// TIA Portal V20 export
// export: Created 2025-12-01T14:57:28.2232406Z, ExportSetting None, DisplayName Totally Integrated Automation Portal, DisplayVersion V20 Update 3, DisplayName TIA Portal Openness, DisplayVersion V20 Update 3, DisplayName TIA Portal Version Control Interface, DisplayVersion V20 Update 3, DisplayName STEP 7 Professional, DisplayVersion V20 Update 3, DisplayName STEP 7 Safety, DisplayVersion V20 Update 2, DisplayName WinCC Basic/Comfort/Advanced, DisplayVersion V20 Update 3, DisplayName WinCC Professional, DisplayVersion V20 Update 3, DisplayName WinCC Unified, DisplayVersion V20 Update 3
FUNCTION_BLOCK "FB605_SalidaFija_Quimarox"   // FB605, LAD
{ S7_Optimized_Access := 'FALSE' }
// stored: AutoNumber false, SetENOAutomatically false
   VAR_INPUT
      MesaSiguiente : UInt;
      MesaDeDescarga : UInt;
      ID_Quimarox : UInt;
      ID_Elemento : UInt;
      EnTension : Bool;
      Termico : Bool;
      pHs_PosicionDescarga : Bool;
      pHs_Protrusion : Bool;
      NXT_PTF : Bool;
      NXT_FTF : Bool;
      V_FILTRO_pHsPresencia : Int;
      Pto_Ajuste_1 : Int;   // Error_protusion
      Pto_Ajuste_2 : Int;   // Paso_A_Lenta
      Pto_Ajuste_3 : Int;   // Error_protusion
   END_VAR
   VAR_OUTPUT
      NXT_DescargaActiva : Bool;   // permiso mesa anterior y avance de la siguiente
      NXT_AVTF : Bool;
      PararElevador : Bool;
      ElevadorEnLenta : Bool;
      Avance_SalidaFija : Bool;
   END_VAR
   VAR
      TMP_EnTension { S7_SetPoint := 'True'} : "FB910_CNT_UHS";
      FILTRO_pHsPresencia { S7_SetPoint := 'True'} : "FB910_CNT_UHS";
      EstadoAsociadoEnMesa { S7_SetPoint := 'True'} : UInt;
      Aux_PeineEnDesCarga : UInt;
      PresenciaEnReset : Bool;
   END_VAR
   VAR_TEMP
      TMP_PeineDeCarga : UInt;
      MesaQuimarox : UInt;
      NumeroUT : UInt;
      EsMesaTL : Bool;
      FILTRO_PosicionDesCarga : Bool;
   END_VAR
BEGIN

NETWORK
TITLE = ERROR - Rearme
/////////////////////////////////////////////////////////////
/////////////////////////////////////////////////////////////
/////////////////////////////////////////////////////////////
// Rearne de Errores
      SET;
      A     "DB902_Estado_ZonaMesa".EstadoMesas[#MesaDeDescarga].Rearme_CBx;
      O     "DB902_Estado_ZonaMesa".EstadoMesas[#MesaDeDescarga].PerReset_CBx;
      R     "DB900_Estado_Mesas".EstadoVI[#MesaDeDescarga].Error_Mx;
      R     "DB900_Estado_Mesas".EstadoVI[#MesaDeDescarga].Err_Protusion;
      R     "DB900_Estado_Mesas".EstadoVI[#MesaDeDescarga].Err_DatosPLC;
      R     "DB900_Estado_Mesas".EstadoVI[#MesaDeDescarga].Err_Termico_E1_E3;
      R     "DB900_Estado_Mesas".EstadoVI[#MesaDeDescarga].Err_Perdida_PHs;


NETWORK
TITLE = RECEP OK DE LA ORDEN -- NO SE UTILIZA
/////////////////////////////////////////////////////////////
/////////////////////////////////////////////////////////////
/////////////////////////////////////////////////////////////
// RECEP OK DE LA ORDEN
      SET;
      AN    "DB841_Recepcion".Mesa[#MesaDeDescarga].Protocolo.Ord_S00;
      AN    "DB841_Recepcion".Mesa[#MesaDeDescarga].Protocolo.Ord_S01;
      AN    "DB841_Recepcion".Mesa[#MesaDeDescarga].Protocolo.Ord_S02;
      AN    "DB841_Recepcion".Mesa[#MesaDeDescarga].Protocolo.Ord_S03;
      NOT;
      =     "DB840_Emision".Mesa[#MesaDeDescarga].Protocolo.RecepOK;



NETWORK
TITLE = HMI - Manual
/////////////////////////////////////////////////////////////
/////////////////////////////////////////////////////////////
/////////////////////////////////////////////////////////////
// Para HMI >>> Manual
      SET;
      O     "DB902_Estado_ZonaMesa".EstadoMesas[#MesaDeDescarga].Manual_CBx;
      =     "DB900_Estado_Mesas".EstadoVI[#MesaDeDescarga].Manual;



NETWORK
TITLE = HMI - Entradas y Salidas de la Mesa
/////////////////////////////////////////////////////////////
/////////////////////////////////////////////////////////////
/////////////////////////////////////////////////////////////
// Entradas
      SET;
      A     #pHs_PosicionDescarga;
      =     "DB900_Estado_Mesas".EstadoVI[#MesaDeDescarga].En_PHS_1;
      SET;
      A     #pHs_Protrusion;
      =     "DB900_Estado_Mesas".EstadoVI[#MesaDeDescarga].En_pHs_Prot1;

      SET;
      A     #Termico;
      =     "DB900_Estado_Mesas".EstadoVI[#MesaDeDescarga].En_Termico1;


// Salidas
      SET;
      A     #Avance_SalidaFija;
      =     "DB900_Estado_Mesas".EstadoVI[#MesaDeDescarga].Sa_Rod_Avance;



NETWORK
TITLE = Comprobacion de que la MESA es de TRACKING
/////////////////////////////////////////////////////////////
/////////////////////////////////////////////////////////////
/////////////////////////////////////////////////////////////
// Comprobar si es una Mesa de Tracking o Routing
      SET;
      A     "DB850_DefinicionMesas".Mesa[#MesaDeDescarga].ConfigMesa.MesaTL;
      =     #EsMesaTL;



REGION Network 6: TMP - Espera En Tension
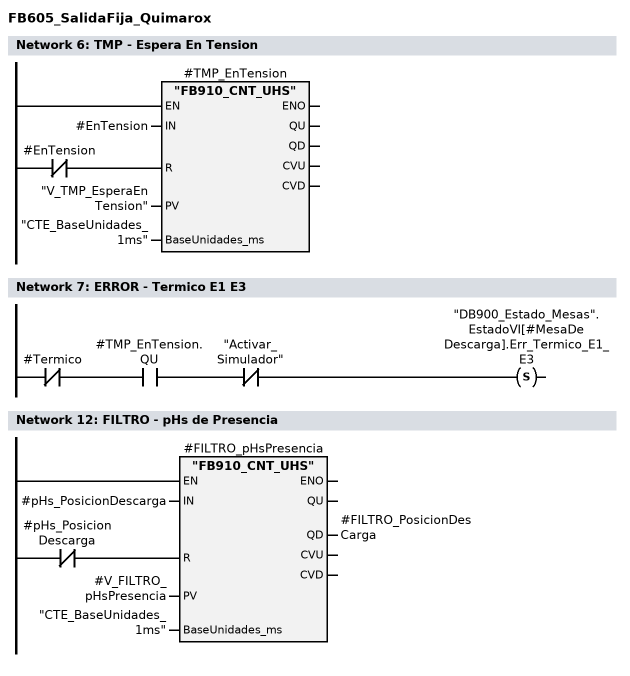
   RUNG wire#powerrail
      #TMP_EnTension(R := wire#w1, IN := #EnTension, PV := "V_TMP_EsperaEnTension", BaseUnidades_ms := "CTE_BaseUnidades_1ms", QU =>, QD =>, CVU =>, CVD =>)
   END_RUNG
   RUNG wire#powerrail
      I_Contact( #EnTension )
   END_RUNG wire#w1
   // the same network as SCL:
   #TMP_EnTension(IN := #EnTension,   // "FB910_CNT_UHS"
                  R := NOT #EnTension,
                  PV := "V_TMP_EsperaEnTension",
                  BaseUnidades_ms := "CTE_BaseUnidades_1ms");
END_REGION

REGION Network 7: ERROR - Termico E1 E3
   RUNG wire#powerrail
      I_Contact( #Termico )
      Contact( #TMP_EnTension.QU )
      I_Contact( "Activar_Simulador" )
      S_Coil( "DB900_Estado_Mesas".EstadoVI[#MesaDeDescarga].Err_Termico_E1_E3 )
   END_RUNG
   // the same network as SCL:
   IF NOT #Termico AND #TMP_EnTension.QU AND NOT "Activar_Simulador" THEN
       "DB900_Estado_Mesas".EstadoVI[#MesaDeDescarga].Err_Termico_E1_E3 := TRUE;
   END_IF;
END_REGION

NETWORK
TITLE = INICIALIZACION Previa
/////////////////////////////////////////////////////////////
/////////////////////////////////////////////////////////////
/////////////////////////////////////////////////////////////
      CLR;
      =     #NXT_DescargaActiva;
      =     #NXT_AVTF;

      CLR;
      =     #ElevadorEnLenta;
      =     #PararElevador;
      =     #Avance_SalidaFija;

      CLR;
      =     "DB900_Estado_Mesas".EstadoVI[#MesaDeDescarga].Etapas_Reset;
      =     "DB900_Estado_Mesas".EstadoVI[#MesaDeDescarga].Etapa_Vacia;
      =     "DB900_Estado_Mesas".EstadoVI[#MesaDeDescarga].Etapa_Cargada;
      =     "DB900_Estado_Mesas".EstadoVI[#MesaDeDescarga].Etapas_Carga_E0;
      =     "DB900_Estado_Mesas".EstadoVI[#MesaDeDescarga].Etapas_Descarga_S3;



NETWORK
TITLE = SISTEMA - Paro Blando
/////////////////////////////////////////////////////////////
/////////////////////////////////////////////////////////////
/////////////////////////////////////////////////////////////
// - Inicializar Variables de PARO BLANDO
      CLR;
      =     "DB900_Estado_Mesas".EstadoVI[#MesaDeDescarga].Paro_Blando;

/////////////////////////////////////////////////////////////
// - Existe PARO BLANDO ???
      SET;
      AN    "DB902_Estado_ZonaMesa".EstadoMesas[#MesaDeDescarga].ParoBlando_CBx;
      JC    NoRealizandose_ParoBlando;

/////////////////////////////////////////////////////////////
// - Fin de PARO BLANDO
      SET;
      =     "DB900_Estado_Mesas".EstadoVI[#MesaDeDescarga].Paro_Blando;


/////////////////////////////////////////////////////////////
/////////////////////////////////////////////////////////////
/////////////////////////////////////////////////////////////
// - Final Tratamiento del PARO BLANDO
NoRealizandose_ParoBlando:NOP   0;



NETWORK
TITLE = SISTEMA - Reset
/////////////////////////////////////////////////////////////
/////////////////////////////////////////////////////////////
/////////////////////////////////////////////////////////////
// -- Inicializar Variables de RESET
      SET;
      AN    "DB902_Estado_ZonaMesa".EstadoMesas[#MesaDeDescarga].PerReset_CBx;
      R     "DB900_Estado_Mesas".EstadoVI[#MesaDeDescarga].Fin_VI;
      R     #PresenciaEnReset;

/////////////////////////////////////////////////////////////
/////////////////////////////////////////////////////////////
/////////////////////////////////////////////////////////////
// - Existe RESET ??
      SET;
      AN    "DB902_Estado_ZonaMesa".EstadoMesas[#MesaDeDescarga].PerReset_CBx;
      JC    NoRealizandose_Reset;

      L     0;  // Estado de La Mesa = 0
      T     #EstadoAsociadoEnMesa;
      SET;
      =     "DB900_Estado_Mesas".EstadoVI[#MesaDeDescarga].Etapas_Reset;

/////////////////////////////////////////////////////////////
/////////////////////////////////////////////////////////////
/////////////////////////////////////////////////////////////
// - Emision de Presencia en caso de Reset
      SET;  // Presencia >>> Reset Total
      A     #pHs_PosicionDescarga;
      A     "DB831_Mesas".Mesas[#MesaDeDescarga].Memorias.M_ResetTotal;
      AN    #PresenciaEnReset;
      JC    Enviar_PresenciaEnResetTotal;

      SET;  // Presencia >>> Reset Parcial
      A     #pHs_PosicionDescarga;
      A     "DB831_Mesas".Mesas[#MesaDeDescarga].Memorias.M_ResetParcial;
      AN    #PresenciaEnReset;
      JC    Enviar_PresenciaEnResetParcial;

      JU    Final_PresenciaEnReset;

// - Presencia en Reset TOTAL >>> Enviar NUUT
Enviar_PresenciaEnResetTotal:NOP   0;
      CALL  "FC723_InsertarUT_EnMesa"
      ( MesaActual := #MesaDeDescarga,
        NumeroUT   := #NumeroUT
      );
      L     132;  // Envio de Nueva UT en RESET
      T     "DB812_UTs_Control".UT[#NumeroUT].EstadoEventoAGenerar;

      SET;  // Ya esta Avisado el JdT
      S     #PresenciaEnReset;

      JU    Final_PresenciaEnReset;

// - Presencia en Reset Parcial >>> Enviar LOCA en Reset Pantalla
Enviar_PresenciaEnResetParcial:NOP   0;
      L     "DB810_ColasMesas".Colas[#MesaDeDescarga].UT_PrimeraMesa;
      T     #NumeroUT;

      L     #NumeroUT;  // Comprobar que Existe UT
      L     0;
      ==I;
      JC    ErrorDatosCargada;

      L     101;  // Envio de LOCA en RESET
      T     "DB812_UTs_Control".UT[#NumeroUT].EstadoEventoAGenerar;

      SET;  // Ya esta Avisado el JdT
      S     #PresenciaEnReset;

      JU    Final_PresenciaEnReset;

// - Final de la Presencia En Reset
Final_PresenciaEnReset:NOP   0;


/////////////////////////////////////////////////////////////
/////////////////////////////////////////////////////////////
/////////////////////////////////////////////////////////////
// - Fin de RESET
      SET;  // Con Presencia de Carga >>> TOTAL
      A(;
      L     "DB810_ColasMesas".Colas[#MesaDeDescarga].UT_PrimeraMesa;
      L     0;
      ==I;
      );
      A     #pHs_PosicionDescarga;
      A     #PresenciaEnReset;
      A     "DB831_Mesas".Mesas[#MesaDeDescarga].Memorias.M_ResetTotal;
      S     "DB900_Estado_Mesas".EstadoVI[#MesaDeDescarga].Fin_VI;

      SET;  // Con Presencia de Carga >>> PARCIAL
      A     #pHs_PosicionDescarga;
      A     #PresenciaEnReset;
      A     "DB831_Mesas".Mesas[#MesaDeDescarga].Memorias.M_ResetParcial;
      S     "DB900_Estado_Mesas".EstadoVI[#MesaDeDescarga].Fin_VI;


      SET;  // Sin Presencia de Carga
      AN    #pHs_PosicionDescarga;
      S     "DB900_Estado_Mesas".EstadoVI[#MesaDeDescarga].Fin_VI;

      BE;

/////////////////////////////////////////////////////////////
/////////////////////////////////////////////////////////////
/////////////////////////////////////////////////////////////
// - Final Tratamiento del RESET
NoRealizandose_Reset:NOP   0;



NETWORK
TITLE = >>>>>>>>>>>>>>>>>>>>>>>>>>>>>>>>>>>>>>>>>>>>>>>>>>>>>>>>>>>>>>>>>>>

REGION Network 12: FILTRO - pHs de Presencia
   RUNG wire#powerrail
      #FILTRO_pHsPresencia(R := wire#w1, IN := #pHs_PosicionDescarga, PV := #V_FILTRO_pHsPresencia, BaseUnidades_ms := "CTE_BaseUnidades_1ms", QU =>, QD => #FILTRO_PosicionDesCarga, CVU =>, CVD =>)
   END_RUNG
   RUNG wire#powerrail
      I_Contact( #pHs_PosicionDescarga )
   END_RUNG wire#w1
   // the same network as SCL:
   #FILTRO_pHsPresencia(IN := #pHs_PosicionDescarga,   // "FB910_CNT_UHS"
                        R := NOT #pHs_PosicionDescarga,
                        PV := #V_FILTRO_pHsPresencia,
                        BaseUnidades_ms := "CTE_BaseUnidades_1ms",
                        QD => #FILTRO_PosicionDesCarga);
END_REGION

NETWORK
TITLE = >>>>>>>>>>>>>>>>>>>>>>>>>>>>>>>>>>>>>>>>>>>>>>>>>>>>>>>>>>>>>>>>>>>

NETWORK
TITLE = DISTRIBUCION >>> Control Etapa Activa
/////////////////////////////////////////////////////////////////////////////////////
/////////////////////////////////////////////////////////////////////////////////////
/////////////////////////////////////////////////////////////////////////////////////
// -- Listado de saltos de programa  >>> Estado
      L     #EstadoAsociadoEnMesa;
      JL    ESTADO_PorDefecto;

      JU    ETAPA_00_EnReset;
      JU    ETAPA_01_EnReposo;
      JU    ETAPA_02_EsperaDesCarga;
      JU    ETAPA_03_DesCargando;
      JU    ETAPA_04_FinalDeDescarga;

      JU    ESTADO_PorDefecto;
      JU    ESTADO_PorDefecto;
      JU    ESTADO_PorDefecto;
      JU    ESTADO_PorDefecto;
      JU    ESTADO_PorDefecto;

      JU    ETAPA_10_ResetCargado_EsperaDesCarga;
      JU    ETAPA_11_ResetCargado_DesCargando;
      JU    ETAPA_12_ResetCargado_FinalDeDescarga;

ESTADO_PorDefecto:JU    FinalFuncion;



NETWORK
TITLE = ETAPA 00 >>> En Reset
/////////////////////////////////////////////////////////////////////////////////////
/////////////////////////////////////////////////////////////////////////////////////
/////////////////////////////////////////////////////////////////////////////////////
ETAPA_00_EnReset:NOP   0;
      SET;
      =     "DB900_Estado_Mesas".EstadoVI[#MesaDeDescarga].Etapas_Reset;

/////////////////////////////////////////////////////////////////////////////////////
// generación de error de protusion
      SET;
      AN    #pHs_Protrusion;
      JC    ErrorProtrusion;


/////////////////////////////////////////////////////////////////////////////////////
// Tiene que estar en Marcha y Sin Error para continuar
      SET;
      AN    "DB902_Estado_ZonaMesa".EstadoMesas[#MesaDeDescarga].Marcha_CBx;
      O     "DB902_Estado_ZonaMesa".EstadoMesas[#MesaDeDescarga].Error_CBx;
      JC    ET00_PararElevador;


/////////////////////////////////////////////////////////////////////////////////////
// Sin Carga
      SET;
      AN    #FILTRO_PosicionDesCarga;
      JC    ET00_IrEtapa_01_EnReposo;

// Con Carga
      SET;
      A     #FILTRO_PosicionDesCarga;
      JC    ET00_IrEtapa_10_ResetCargado_EsperaDesCarga;
      BE;


/////////////////////////////////////////////////////////////////////////////////////
/////////////////////////////////////////////////////////////////////////////////////
/////////////////////////////////////////////////////////////////////////////////////
ET00_PararElevador:NOP   0;
      SET;
      =     #PararElevador;
      BE;


/////////////////////////////////////////////////////////////////////////////////////
/////////////////////////////////////////////////////////////////////////////////////
/////////////////////////////////////////////////////////////////////////////////////
ET00_IrEtapa_01_EnReposo:NOP   0;
      L     1;
      T     #EstadoAsociadoEnMesa;
      JU    ETAPA_01_EnReposo;


/////////////////////////////////////////////////////////////////////////////////////
/////////////////////////////////////////////////////////////////////////////////////
/////////////////////////////////////////////////////////////////////////////////////
ET00_IrEtapa_10_ResetCargado_EsperaDesCarga:NOP   0;
      SET;  // No existe UT >>> Error de Datos
      A(;
      L     "DB810_ColasMesas".Colas[#MesaDeDescarga].UT_PrimeraMesa;
      L     0;
      ==I;
      );
      AN    #EsMesaTL;
      JC    ErrorDatosCargada;

      L     10;
      T     #EstadoAsociadoEnMesa;
      JU    ETAPA_10_ResetCargado_EsperaDesCarga;



NETWORK
TITLE = ETAPA 01 >>> En Reposo
/////////////////////////////////////////////////////////////////////////////////////
/////////////////////////////////////////////////////////////////////////////////////
/////////////////////////////////////////////////////////////////////////////////////
// comprobamos si tenemos que parar el elevador por seguridad
ETAPA_01_EnReposo:NOP   0;
      SET;
      =     "DB900_Estado_Mesas".EstadoVI[#MesaDeDescarga].Etapa_Vacia;


/////////////////////////////////////////////////////////////////////////////////////
// Comprobar si hay algo en la Mesa
      SET;
      A     #FILTRO_PosicionDesCarga;
      JC    ET01_IrEtapa_02_SalidaDePeine;

/////////////////////////////////////////////////////////////////////////////////////
/////////////////////////////////////////////////////////////////////////////////////
/////////////////////////////////////////////////////////////////////////////////////
// error protusion, hay algo y en ese momento no debería haber nada
      SET;
      AN    "DB602_ElementosQuimarox".Quimarox[#ID_Quimarox].Elementos[#ID_Elemento].Hay_Carrier_en_ventana;
      A(;
      ON    #pHs_Protrusion;
      O     #FILTRO_PosicionDesCarga;
      );
      JC    ErrorProtrusion;

/////////////////////////////////////////////////////////////////////////////////////
// error protusion, hay algo y en ese momento no debería haber nada
      SET;
      A     "DB602_ElementosQuimarox".Quimarox[#ID_Quimarox].Elementos[#ID_Elemento].Hay_Carrier_en_ventana;
      A(;
      L     "DB602_ElementosQuimarox".Quimarox[#ID_Quimarox].Elementos[#ID_Elemento].Avance_carrier;
      L     #Pto_Ajuste_1;
      <=I;
      );
      A(;
      ON    #pHs_Protrusion;
      O     #FILTRO_PosicionDesCarga;
      );
      JC    ErrorProtrusion;


/////////////////////////////////////////////////////////////////////////////////////
/////////////////////////////////////////////////////////////////////////////////////
/////////////////////////////////////////////////////////////////////////////////////
// No deberia estar en este Estado, ha pasado sin carga


/////////////////////////////////////////////////////////////////////////////////////
// Parar por seguridad
      SET;
      A     "DB602_ElementosQuimarox".Quimarox[#ID_Quimarox].Elementos[#ID_Elemento].Hay_Carrier_en_ventana;
      A(;
      L     "DB602_ElementosQuimarox".Quimarox[#ID_Quimarox].Elementos[#ID_Elemento].Avance_carrier;  // #datos_elemento_Tmp.Avance_carrier
      L     #Pto_Ajuste_3;
      >=I;
      );
      A(;
      ON    #pHs_Protrusion;
      O     #FILTRO_PosicionDesCarga;
      );
      JC    ET01_PararElevador;


/////////////////////////////////////////////////////////////////////////////////////
// Lenta por seguridad
      SET;
      A     "DB602_ElementosQuimarox".Quimarox[#ID_Quimarox].Elementos[#ID_Elemento].Hay_Carrier_en_ventana;
      A(;
      L     "DB602_ElementosQuimarox".Quimarox[#ID_Quimarox].Elementos[#ID_Elemento].Avance_carrier;  // #datos_elemento_Tmp.Avance_carrier
      L     #Pto_Ajuste_2;
      >=I;
      );
      A(;
      ON    #pHs_Protrusion;
      O     #FILTRO_PosicionDesCarga;
      );
      JC    ET01_VelocidadLenta;

/////////////////////////////////////////////////////////////////////////////////////
// Final de Estado
      BE;


/////////////////////////////////////////////////////////////////////////////////////
/////////////////////////////////////////////////////////////////////////////////////
/////////////////////////////////////////////////////////////////////////////////////
ET01_PararElevador:NOP   0;
      SET;
      =     #PararElevador;

      BE;

/////////////////////////////////////////////////////////////////////////////////////
/////////////////////////////////////////////////////////////////////////////////////
/////////////////////////////////////////////////////////////////////////////////////
ET01_VelocidadLenta:NOP   0;
      SET;
      =     #ElevadorEnLenta;
      BE;


/////////////////////////////////////////////////////////////////////////////////////
/////////////////////////////////////////////////////////////////////////////////////
/////////////////////////////////////////////////////////////////////////////////////
ET01_IrEtapa_02_SalidaDePeine:NOP   0;
      L     "DB602_ElementosQuimarox".Quimarox[#ID_Quimarox].Elementos[#ID_Elemento].Numero_carrier;
      T     #Aux_PeineEnDesCarga;

// Emision del Evento del Quimarox
      L     "CTE_Evento_QDES";
      T     "DB601_PeinesQuimarox".Quimarox[#ID_Quimarox].vagon[#Aux_PeineEnDesCarga].EventoAGenerar;
      L     #MesaDeDescarga;
      L     "CTE_OffsetMesa";
      +I;
      T     "DB601_PeinesQuimarox".Quimarox[#ID_Quimarox].vagon[#Aux_PeineEnDesCarga].Mesa_descarga;

/////////////////////////////////////////////////////////////////////////////////////
/////////////////////////////////////////////////////////////////////////////////////
/////////////////////////////////////////////////////////////////////////////////////
// Comprobar Tipo de Mesa
      SET;
      A     #EsMesaTL;
      JC    ET01_Final_RecogerDatosDelPeine;

/////////////////////////////////////////////////////////////////////////////////////
// TRACKING - INICIO - Recoger Datos del Peine
      SET;
      L     "DB601_PeinesQuimarox".Quimarox[#ID_Quimarox].vagon[#Aux_PeineEnDesCarga].DatosCarga.Mckey;
      L     0;
      ==D;
      JC    ET01_TRACKING_CrearNueva_UT;
      JU    ET01_TRACKING_Crear_UT;


/////////////////////////////////////////////////////////////////////////////////////
// TRAKING - NuevaUT en la Mesa
ET01_TRACKING_Crear_UT:NOP   0;
      CALL  "FC721_CrearUT_EnMesa"
      ( McKey      := "DB601_PeinesQuimarox".Quimarox[#ID_Quimarox].vagon[#Aux_PeineEnDesCarga].DatosCarga.Mckey,
        MesaActual := #MesaDeDescarga,
        NumeroUT   := #NumeroUT
      );

      L     100;  // Emitir evento LOCA
      T     "DB812_UTs_Control".UT[#NumeroUT].EstadoEventoAGenerar;

      L     "DB601_PeinesQuimarox".Quimarox[#ID_Quimarox].vagon[#Aux_PeineEnDesCarga].DatosCarga.MesaDestino;
      T     "DB812_UTs_Control".UT[#NumeroUT].MesaDestino;
      T     "DB812_UTs_Control".UT[#NumeroUT].MesaIntermedia;
      T     "DB813_UTs_Ruta".UT[#NumeroUT].Ruta[0];

      JU    ET01_Final_RecogerDatosDelPeine;


/////////////////////////////////////////////////////////////////////////////////////
// TRAKING - NuevaUT en la Mesa
ET01_TRACKING_CrearNueva_UT:NOP   0;
      JU    ET01_Final_RecogerDatosDelPeine;


/////////////////////////////////////////////////////////////////////////////////////
// Final de la Recogida de Datos del Peine
ET01_Final_RecogerDatosDelPeine:NOP   0;
      L     2;
      T     #EstadoAsociadoEnMesa;
      JU    ETAPA_02_EsperaDesCarga;



NETWORK
TITLE = ETAPA 02 >>> Espera de Inicio de DesCarga
/////////////////////////////////////////////////////////////////////////////////////
/////////////////////////////////////////////////////////////////////////////////////
/////////////////////////////////////////////////////////////////////////////////////
ETAPA_02_EsperaDesCarga:NOP   0;
      SET;
      =     "DB900_Estado_Mesas".EstadoVI[#MesaDeDescarga].Etapa_Cargada;


/////////////////////////////////////////////////////////////////////////////////////
      SET;
      =     #NXT_AVTF;

/////////////////////////////////////////////////////////////////////////////////////
// comprobamos si tenemos que pasar al estado de descarga activa
      SET;
      A     #NXT_PTF;
      JC    ET02_IrEtapa_03_DesCargando;


/////////////////////////////////////////////////////////////////////////////////////
/////////////////////////////////////////////////////////////////////////////////////
/////////////////////////////////////////////////////////////////////////////////////
// error protusion, hay algo y en ese momento no debería haber nada
      SET;
      AN    "DB602_ElementosQuimarox".Quimarox[#ID_Quimarox].Elementos[#ID_Elemento].Hay_Carrier_en_ventana;
      A(;
      ON    #pHs_Protrusion;
      O     #FILTRO_PosicionDesCarga;
      );
      JC    ErrorProtrusion;


/////////////////////////////////////////////////////////////////////////////////////
// error protusion, hay algo y en ese momento no debería haber nada, YA DEBERIA HABER PASADO ESTE PUNTO
      SET;
      A     "DB602_ElementosQuimarox".Quimarox[#ID_Quimarox].Elementos[#ID_Elemento].Hay_Carrier_en_ventana;
      A(;
      L     "DB602_ElementosQuimarox".Quimarox[#ID_Quimarox].Elementos[#ID_Elemento].Avance_carrier;
      L     #Pto_Ajuste_1;
      <=I;
      );
      A(;
      ON    #pHs_Protrusion;
      O     #FILTRO_PosicionDesCarga;
      );
      JC    ErrorProtrusion;

/////////////////////////////////////////////////////////////////////////////////////
/// LIMITE DE LA DESCARGA --- PARAR ELEVADOR
      SET;
      A     "DB602_ElementosQuimarox".Quimarox[#ID_Quimarox].Elementos[#ID_Elemento].Hay_Carrier_en_ventana;
      A(;
      L     "DB602_ElementosQuimarox".Quimarox[#ID_Quimarox].Elementos[#ID_Elemento].Avance_carrier;  // #datos_elemento_Tmp.Avance_carrier
      L     #Pto_Ajuste_3;
      >=I;
      );
      A(;
      ON    #pHs_Protrusion;
      O     #FILTRO_PosicionDesCarga;
      );
      JC    ET02_PararElevador;


/////////////////////////////////////////////////////////////////////////////////////
// comprobación de rango para paso a lenta por seguridad
/// ESTA LLEGANDO AL LIMITE DE LA DESCARGA --- LENTO ELEVADOR
      SET;
      A     "DB602_ElementosQuimarox".Quimarox[#ID_Quimarox].Elementos[#ID_Elemento].Hay_Carrier_en_ventana;
      A(;
      L     "DB602_ElementosQuimarox".Quimarox[#ID_Quimarox].Elementos[#ID_Elemento].Avance_carrier;  // #datos_elemento_Tmp.Avance_carrier
      L     #Pto_Ajuste_2;
      >=I;
      );
      A(;
      ON    #pHs_Protrusion;
      O     #FILTRO_PosicionDesCarga;
      );
      JC    ET02_VelocidadLenta;

/////////////////////////////////////////////////////////////////////////////////////
// Perdida de Presencia de Carga antes de iniciar la descarga
      SET;
      AN    #FILTRO_PosicionDesCarga;
      JC    ErrorPerdidaPresencia;

/////////////////////////////////////////////////////////////////////////////////////
// Final de Estado
      BE;


/////////////////////////////////////////////////////////////////////////////////////
/////////////////////////////////////////////////////////////////////////////////////
/////////////////////////////////////////////////////////////////////////////////////
ET02_PararElevador:NOP   0;
      SET;
      =     #PararElevador;
      BE;

/////////////////////////////////////////////////////////////////////////////////////
/////////////////////////////////////////////////////////////////////////////////////
/////////////////////////////////////////////////////////////////////////////////////
ET02_VelocidadLenta:NOP   0;
      SET;
      =     #ElevadorEnLenta;
      BE;


/////////////////////////////////////////////////////////////////////////////////////
/////////////////////////////////////////////////////////////////////////////////////
/////////////////////////////////////////////////////////////////////////////////////
ET02_IrEtapa_03_DesCargando:NOP   0;
      L     3;
      T     #EstadoAsociadoEnMesa;
      JU    ETAPA_03_DesCargando;




NETWORK
TITLE = ETAPA 03 >>> DesCargando
/////////////////////////////////////////////////////////////////////////////////////
/////////////////////////////////////////////////////////////////////////////////////
/////////////////////////////////////////////////////////////////////////////////////
// controlamos el proceso de descarga.
ETAPA_03_DesCargando:NOP   0;
      SET;
      =     "DB900_Estado_Mesas".EstadoVI[#MesaDeDescarga].Etapas_Descarga_S3;


/////////////////////////////////////////////////////////////////////////////////////
      SET;
      =     #NXT_DescargaActiva;
      =     #NXT_AVTF;

      SET;
      A     #NXT_PTF;
      =     #Avance_SalidaFija;


/////////////////////////////////////////////////////////////////////////////////////
/////////////////////////////////////////////////////////////////////////////////////
/////////////////////////////////////////////////////////////////////////////////////
      SET;  // Fin de la DesCarga
      AN    #FILTRO_PosicionDesCarga;
      A     #pHs_Protrusion;
      A     #NXT_FTF;
      JC    ET03_IrEtapa_04_FinalDeDesCarga;


/////////////////////////////////////////////////////////////////////////////////////
/////////////////////////////////////////////////////////////////////////////////////
/////////////////////////////////////////////////////////////////////////////////////
// error protusion, hay algo y en ese momento no debería haber nada
      SET;
      AN    "DB602_ElementosQuimarox".Quimarox[#ID_Quimarox].Elementos[#ID_Elemento].Hay_Carrier_en_ventana;  //#datos_elemento_Tmp.Hay_Carrier_en_ventana
      A(;
      O     #FILTRO_PosicionDesCarga;
      ON    #pHs_Protrusion;
      );
      JC    ErrorProtrusion;

/////////////////////////////////////////////////////////////////////////////////////
// error protusion, hay algo y en ese momento no debería haber nada, YA DEBERIA HABER PASADO ESTE PUNTO
      SET;
      A     "DB602_ElementosQuimarox".Quimarox[#ID_Quimarox].Elementos[#ID_Elemento].Hay_Carrier_en_ventana;
      A(;
      L     "DB602_ElementosQuimarox".Quimarox[#ID_Quimarox].Elementos[#ID_Elemento].Avance_carrier;
      L     #Pto_Ajuste_1;
      <=I;
      );
      A(;
      ON    #pHs_Protrusion;
      O     #FILTRO_PosicionDesCarga;
      );
      JC    ErrorProtrusion;

/////////////////////////////////////////////////////////////////////////////////////
/// LIMITE DE LA DESCARGA --- PARAR ELEVADOR
      SET;
      A     "DB602_ElementosQuimarox".Quimarox[#ID_Quimarox].Elementos[#ID_Elemento].Hay_Carrier_en_ventana;
      A(;
      L     "DB602_ElementosQuimarox".Quimarox[#ID_Quimarox].Elementos[#ID_Elemento].Avance_carrier;  // #datos_elemento_Tmp.Avance_carrier
      L     #Pto_Ajuste_3;
      >=I;
      );
      A(;
      ON    #pHs_Protrusion;
      O     #FILTRO_PosicionDesCarga;
      );
      JC    ET03_PararElevador;


/////////////////////////////////////////////////////////////////////////////////////
// comprobación de rango para paso a lenta por seguridad
/// ESTA LLEGANDO AL LIMITE DE LA DESCARGA --- PARAR ELEVADOR
      SET;
      A     "DB602_ElementosQuimarox".Quimarox[#ID_Quimarox].Elementos[#ID_Elemento].Hay_Carrier_en_ventana;  //  #datos_elemento_Tmp.Hay_Carrier_en_ventana
      A(;
      L     "DB602_ElementosQuimarox".Quimarox[#ID_Quimarox].Elementos[#ID_Elemento].Avance_carrier;  // #datos_elemento_Tmp.Avance_carrier
      L     #Pto_Ajuste_2;
      >=I;
      );
      JC    ET03_VelocidadLenta;

/////////////////////////////////////////////////////////////////////////////////////
// Final de Estado
      BE;


/////////////////////////////////////////////////////////////////////////////////////
/////////////////////////////////////////////////////////////////////////////////////
/////////////////////////////////////////////////////////////////////////////////////
ET03_PararElevador:NOP   0;
      SET;
      =     #PararElevador;
      BE;

/////////////////////////////////////////////////////////////////////////////////////
/////////////////////////////////////////////////////////////////////////////////////
/////////////////////////////////////////////////////////////////////////////////////
ET03_VelocidadLenta:NOP   0;
      SET;
      =     #ElevadorEnLenta;
      BE;


/////////////////////////////////////////////////////////////////////////////////////
/////////////////////////////////////////////////////////////////////////////////////
/////////////////////////////////////////////////////////////////////////////////////
ET03_IrEtapa_04_FinalDeDesCarga:NOP   0;
      L     4;
      T     #EstadoAsociadoEnMesa;
      JU    ETAPA_04_FinalDeDescarga;



NETWORK
TITLE = ETAPA 04 >>> Final De Descarga >>>> PASA LOS DATOS
/////////////////////////////////////////////////////////////////////////////////////
/////////////////////////////////////////////////////////////////////////////////////
/////////////////////////////////////////////////////////////////////////////////////
ETAPA_04_FinalDeDescarga:NOP   0;
      SET;
      =     "DB900_Estado_Mesas".EstadoVI[#MesaDeDescarga].Etapas_Descarga_S3;


/////////////////////////////////////////////////////////////////////////////////////
      CLR;
      =     #NXT_DescargaActiva;
      =     #NXT_AVTF;
      =     #ElevadorEnLenta;
      =     #PararElevador;
      =     #Avance_SalidaFija;


/////////////////////////////////////////////////////////////////////////////////////
/////////////////////////////////////////////////////////////////////////////////////
/////////////////////////////////////////////////////////////////////////////////////
      JU    ET04_IrEtapa_01_EnReposo;


/////////////////////////////////////////////////////////////////////////////////////
/////////////////////////////////////////////////////////////////////////////////////
/////////////////////////////////////////////////////////////////////////////////////
ET04_IrEtapa_01_EnReposo:NOP   0;
      L     1;
      T     #EstadoAsociadoEnMesa;
      JU    ETAPA_01_EnReposo;



NETWORK
TITLE = >>>>>>>>>>>>>>>>>>>>>>>>>>>>>>>>>>>>>>>>>>>>>>>>>>>>>>>>>>>>>>>>>>>

NETWORK
TITLE = ETAPA 10 >>> RESET CARGADO >>> Espera de Inicio de DesCarga
/////////////////////////////////////////////////////////////////////////////////////
/////////////////////////////////////////////////////////////////////////////////////
/////////////////////////////////////////////////////////////////////////////////////
ETAPA_10_ResetCargado_EsperaDesCarga:NOP   0;
      SET;
      =     "DB900_Estado_Mesas".EstadoVI[#MesaDeDescarga].Etapas_Reset;


/////////////////////////////////////////////////////////////////////////////////////
// error de protusion
      SET;
      AN    #pHs_Protrusion;
      JC    ErrorProtrusion;


/////////////////////////////////////////////////////////////////////////////////////
/////////////////////////////////////////////////////////////////////////////////////
/////////////////////////////////////////////////////////////////////////////////////
      SET;
      =     #PararElevador;
      =     #NXT_AVTF;

/////////////////////////////////////////////////////////////////////////////////////
      SET;
      A     #NXT_PTF;
      JC    ET10_IrEtapa_11_ResetCargado_DesCargando;


/////////////////////////////////////////////////////////////////////////////////////
// Perdida de Presencia de Carga antes de iniciar la descarga
      SET;
      AN    #FILTRO_PosicionDesCarga;
      JC    ErrorPerdidaPresencia;

/////////////////////////////////////////////////////////////////////////////////////
// Final de Estado
      BE;



/////////////////////////////////////////////////////////////////////////////////////
/////////////////////////////////////////////////////////////////////////////////////
/////////////////////////////////////////////////////////////////////////////////////
ET10_IrEtapa_11_ResetCargado_DesCargando:NOP   0;
      L     11;
      T     #EstadoAsociadoEnMesa;
      JU    ETAPA_11_ResetCargado_DesCargando;




NETWORK
TITLE = ETAPA 11 >>> RESET CARGADO >>> DesCargando
/////////////////////////////////////////////////////////////////////////////////////
/////////////////////////////////////////////////////////////////////////////////////
/////////////////////////////////////////////////////////////////////////////////////
// controlamos el proceso de descarga.
ETAPA_11_ResetCargado_DesCargando:NOP   0;
      SET;
      =     "DB900_Estado_Mesas".EstadoVI[#MesaDeDescarga].Etapas_Descarga_S3;
      =     "DB900_Estado_Mesas".EstadoVI[#MesaDeDescarga].Etapas_Reset;


/////////////////////////////////////////////////////////////////////////////////////
      SET;
      =     #PararElevador;
      =     #NXT_DescargaActiva;
      =     #NXT_AVTF;

      SET;
      A     #NXT_PTF;
      =     #Avance_SalidaFija;


/////////////////////////////////////////////////////////////////////////////////////
/////////////////////////////////////////////////////////////////////////////////////
/////////////////////////////////////////////////////////////////////////////////////
      SET;  // Fin de la DesCarga
      AN    #FILTRO_PosicionDesCarga;
      A     #pHs_Protrusion;
      A     #NXT_FTF;
      JC    ET11_IrEtapa_12_ResetCargado_FinalDeDesCarga;


/////////////////////////////////////////////////////////////////////////////////////
// Final de Estado
      BE;


/////////////////////////////////////////////////////////////////////////////////////
/////////////////////////////////////////////////////////////////////////////////////
/////////////////////////////////////////////////////////////////////////////////////
ET11_IrEtapa_12_ResetCargado_FinalDeDesCarga:NOP   0;
      L     12;
      T     #EstadoAsociadoEnMesa;
      JU    ETAPA_12_ResetCargado_FinalDeDescarga;



NETWORK
TITLE = ETAPA 12 >>> RESET CARGADO >>> Final De Descarga >>>> PASA LOS DATOS
/////////////////////////////////////////////////////////////////////////////////////
/////////////////////////////////////////////////////////////////////////////////////
/////////////////////////////////////////////////////////////////////////////////////
ETAPA_12_ResetCargado_FinalDeDescarga:NOP   0;
      SET;
      =     "DB900_Estado_Mesas".EstadoVI[#MesaDeDescarga].Etapas_Descarga_S3;
      =     "DB900_Estado_Mesas".EstadoVI[#MesaDeDescarga].Etapas_Reset;

/////////////////////////////////////////////////////////////////////////////////////
      SET;
      =     #PararElevador;

      CLR;
      =     #NXT_DescargaActiva;
      =     #NXT_AVTF;
      =     #Avance_SalidaFija;

/////////////////////////////////////////////////////////////////////////////////////
/////////////////////////////////////////////////////////////////////////////////////
/////////////////////////////////////////////////////////////////////////////////////
      JU    ET12_IrEtapa_01_ResetCargado_EnReposo;


/////////////////////////////////////////////////////////////////////////////////////
/////////////////////////////////////////////////////////////////////////////////////
/////////////////////////////////////////////////////////////////////////////////////
ET12_IrEtapa_01_ResetCargado_EnReposo:NOP   0;
      L     1;
      T     #EstadoAsociadoEnMesa;
      JU    ETAPA_01_EnReposo;



NETWORK
TITLE = >>>>>>>>>>>>>>>>>>>>>>>>>>>>>>>>>>>>>>>>>>>>>>>>>>>>>>>>>>>>>>>>>>>

NETWORK
TITLE = ERRRORES DE LA MESA >>> Activacion
/////////////////////////////////////////////////////////////////////////////////////
/////////////////////////////////////////////////////////////////////////////////////
/////////////////////////////////////////////////////////////////////////////////////
ErrorProtrusion:NOP   0;
      SET;
      =     #PararElevador;
      =     "DB900_Estado_Mesas".EstadoVI[#MesaDeDescarga].Err_Protusion;
      S     "DB900_Estado_Mesas".EstadoVI[#MesaDeDescarga].Error_Mx;
      BE;


/////////////////////////////////////////////////////////////////////////////////////
/////////////////////////////////////////////////////////////////////////////////////
/////////////////////////////////////////////////////////////////////////////////////
ErrorPerdidaPresencia:NOP   0;  // error de Perdida de Presencia
      SET;
      =     "DB900_Estado_Mesas".EstadoVI[#MesaDeDescarga].Err_Perdida_PHs;
      S     "DB900_Estado_Mesas".EstadoVI[#MesaDeDescarga].Error_Mx;
      =     #PararElevador;
      BE;


/////////////////////////////////////////////////////////////////////////////////////
/////////////////////////////////////////////////////////////////////////////////////
/////////////////////////////////////////////////////////////////////////////////////
ErrorDatosCargada:NOP   0;  // error en la carga
      SET;
      =     "DB900_Estado_Mesas".EstadoVI[#MesaDeDescarga].Err_DatosPLC;
      S     "DB900_Estado_Mesas".EstadoVI[#MesaDeDescarga].Error_Mx;
      =     #PararElevador;
      BE;



NETWORK
TITLE = FINAL DE LA FUNCION
/////////////////////////////////////////////////////////////////////////////////////
/////////////////////////////////////////////////////////////////////////////////////
/////////////////////////////////////////////////////////////////////////////////////
FinalFuncion:BE;


END_FUNCTION_BLOCK
